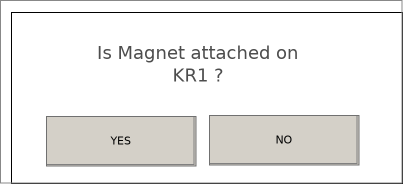
VISUALIZATION MSG_EOAT  // 403x184
    RoundedRectangle (11,12 392x172)
    Button (46,116 150x50), "YES"
        OnMouseClick: execute { GVL.KR1_EOAT_FILL:= TRUE; GVL.KR1_EOAT_SUCTION:= FALSE; }
        OnMouseClick: CloseDialog Dialog=MSG_EOAT, Result=Yes, NumpadKeypadSet=True
    Button (209,115 150x50), "NO"
        OnMouseClick: execute { GVL.KR1_EOAT_FILL:= FALSE; }
        OnMouseClick: CloseDialog Dialog=MSG_EOAT, Result=No, NumpadKeypadSet=True
    Label (80,20 236x88), "Is Magnet attached on KR1 ?"
END_VISUALIZATION

(* stored: Version 1.1.0.1, ProductVersion 3.1.4024.12
   Visu MSG_EOAT: Id {aac8cffe-b23d-460a-9c05-fb0383771a34} *)
